// TIA Portal project "PA_test" (V13)

(* hardware
DEVICE "S7300/ET200M station_1"  S7-300 station
   slot 0: "Rail_0"  Rail  6ES7 390-1***0-0AA0
   slot 1: "PS 307 5A_1"  PS 307 5A  6ES7 307-1EA01-0AA0
   slot 2: "PLC-243"  CPU 314C-2 PN/DP  6ES7 314-6EH04-0AB0  V3.3
      slot 2: "PROFINET interface_1"  PN-IO
         slot 1: "Port_1"  Port
         slot 2: "Port_2"  Port
      slot 5: "DI 24/DO 16_1"  DI24/DO16
      slot 6: "AI 5/AO 2_1"  AI5/AO2
      slot 7: "Count_1"  Counter
      slot 8: "Positioning_1"  Positioning
   slot 4: "DI 16x24VDC_1"  DI16 x 24VDC  6ES7 321-1BH02-0AA0
DEVICE "PC station"  SIMATIC PC station
   slot 0: "PC station"  Rail  SIMATIC PC-Station  V1.0
      slot 125: "Stationmanager"  Station_Manager  V6.0.4
   slot 1: "IE general_1"  IE General  IE_CP  V8.2.0
   slot 3: "HMI_RT_1"  WinCC RT Advanced  6AV2 104-0xxxx-xxxx  13.0.1.0
      slot 33792: "Host interface"  Host interface
*)

// ===== PLC "PLC-243"  CPU 314C-2 PN/DP =====

VAR_GLOBAL   // PLC tag table "Default tag table"
   "crna_levo_zgoraj" AT %I1.4 : Bool;
   "crna_desno_zgoraj" AT %I1.6 : Bool;
   "rdeca_levo_zgoraj" AT %Q1.4 : Bool;
   "kljuc" AT %I1.2 : Bool;
   "rdeca_desno_zgoraj" AT %Q1.6 : Bool;
   "stanje" AT %M0.0 : Bool;
   "zelena_tipka" AT %I1.3 : Bool;
   "dvig_smer" AT %Q0.4 : Bool;
   "crna_levo_spodaj" AT %I1.5 : Bool;
   "crna_desno_spodaj" AT %I1.7 : Bool;
   "stevec_trenutno_s" AT %MW4 : Int;
   "miza_premik" AT %Q0.1 : Bool;
   "miza_smer" AT %Q0.0 : Bool;
   "roka_premik" AT %Q0.3 : Bool;
   "roka_smer" AT %Q0.2 : Bool;
   "dvig_premik" AT %Q0.5 : Bool;
   "prijemalo_smer" AT %Q0.6 : Bool;
   "prijemalo_premik" AT %Q0.7 : Bool;
   "koncno_stikalo_miza" AT %I0.0 : Bool;
   "koncno_stikalo_roka" AT %I0.2 : Bool;
   "bit_vrednost" AT %M0.4 : Bool;
   "stevec_impulza_miza" AT %MW10 : Int;
   "impulz_miza" AT %I0.1 : Bool;
   "impulz_roka" AT %I0.3 : Bool;
   "stevec_impulza_roka" AT %MW12 : Int;
   "stevec_impulza_dvig" AT %MW14 : Int;
   "koncno_stikalo_dvig" AT %I0.4 : Bool;
   "impulz_dvig" AT %I0.5 : Bool;
   "koncno_stikalo_prijemalo" AT %I0.6 : Bool;
   "impulz_prijemalo" AT %I0.7 : Bool;
   "stevec_impulza_prijemalo" AT %MW16 : Int;
   "avto_miza_CW" AT %M5.5 : Bool;
   "avto_miza_CCW" AT %M5.6 : Bool;
   "konec_miza" AT %M7.0 : Bool;
   "avto_roka_CW" AT %M5.7 : Bool;
   "avto_roka_CCW" AT %M6.0 : Bool;
   "konec_roka" AT %M6.1 : Bool;
   "avto_dvig_CW" AT %M6.2 : Bool;
   "avto_dvig_CCW" AT %M6.3 : Bool;
   "konec_dvig" AT %M6.4 : Bool;
   "avto_prijemalo_CW" AT %M6.5 : Bool;
   "avto_prijemalo_CCW" AT %M6.6 : Bool;
   "konec_prijemalo" AT %M6.7 : Bool;
   "miza_enable" AT %M7.1 : Bool;
   "miza_koliko" AT %MW8 : Int;
   "roka_koliko" AT %MW18 : Int;
   "dvig_koliko" AT %MW20 : Int;
   "prijemalo_koliko" AT %MW22 : Int;
   "roka_enable" AT %M7.2 : Bool;
   "dvig_enable" AT %M7.3 : Bool;
   "prijemalo_enable" AT %M7.4 : Bool;
   "upravljanje_avtomatov_enable" AT %M24.0 : Bool;
   "rumena_levo_spodaj" AT %Q1.5 : Bool;
   "rumena_desno_spodaj" AT %Q1.7 : Bool;
   "recept" AT %M24.1 : Bool;
END_VAR

TYPE "UDT_lokacija"
   STRUCT
      ID_lokacije : Int;
      miza_lokacija : Int;
      izteg_lokacija : Int;
      stisk_lokacija : Int;
      dvig_lokacija : Int;
   END_STRUCT;
END_TYPE

DATA_BLOCK "stevec_izbira_motorja_DB"   // DB1
{ S7_Optimized_Access := 'FALSE' }
VERSION : 0.1
// stored: InstanceOfName stevec_izbira_motorja
"stevec_izbira_motorja"
BEGIN
END_DATA_BLOCK

DATA_BLOCK "motor_roka"   // DB2
{ S7_Optimized_Access := 'FALSE' }
VERSION : 0.1
// stored: InstanceOfName motor1
"motor1"
BEGIN
END_DATA_BLOCK

DATA_BLOCK "motor1_DB"   // DB3
{ S7_Optimized_Access := 'FALSE' }
VERSION : 0.1
// stored: InstanceOfName motor1
"motor1"
BEGIN
END_DATA_BLOCK

DATA_BLOCK "avtomat_miza_DB"   // DB4
{ S7_Optimized_Access := 'FALSE' }
VERSION : 0.1
// stored: InstanceOfName avtomat_miza
"avtomat_miza"
BEGIN
END_DATA_BLOCK

DATA_BLOCK "Lokacije"   // DB5
{ S7_Optimized_Access := 'FALSE' }
VERSION : 0.1
   VAR
      Lokacija : Array[0..7] of "UDT_lokacija";
   END_VAR
BEGIN
END_DATA_BLOCK

DATA_BLOCK "motor_miza"   // DB6
{ S7_Optimized_Access := 'FALSE' }
VERSION : 0.1
// stored: InstanceOfName motor1
"motor1"
BEGIN
END_DATA_BLOCK

DATA_BLOCK "motor_dvig"   // DB8
{ S7_Optimized_Access := 'FALSE' }
VERSION : 0.1
// stored: InstanceOfName motor1
"motor1"
BEGIN
END_DATA_BLOCK

DATA_BLOCK "motor_prijemalo"   // DB9
{ S7_Optimized_Access := 'FALSE' }
VERSION : 0.1
// stored: InstanceOfName motor1
"motor1"
BEGIN
END_DATA_BLOCK

DATA_BLOCK "avtomat_roka_DB"   // DB10
{ S7_Optimized_Access := 'FALSE' }
VERSION : 0.1
// stored: InstanceOfName avtomat_roka
"avtomat_roka"
BEGIN
END_DATA_BLOCK

DATA_BLOCK "avtomat_dvig_DB"   // DB11
{ S7_Optimized_Access := 'FALSE' }
VERSION : 0.1
// stored: InstanceOfName avtomat_dvig
"avtomat_dvig"
BEGIN
END_DATA_BLOCK

DATA_BLOCK "avtomat_prijemalo_DB"   // DB12
{ S7_Optimized_Access := 'FALSE' }
VERSION : 0.1
// stored: InstanceOfName avtomat_prijemalo
"avtomat_prijemalo"
BEGIN
END_DATA_BLOCK

DATA_BLOCK "upravljanje_avtomatov_DB"   // DB13
{ S7_Optimized_Access := 'FALSE' }
VERSION : 0.1
// stored: InstanceOfName upravljanje_avtomatov
"upravljanje_avtomatov"
BEGIN
END_DATA_BLOCK

DATA_BLOCK "zunanji_krmilnik_DB"   // DB14
{ S7_Optimized_Access := 'FALSE' }
VERSION : 0.1
// stored: InstanceOfName zunanji_krmilnik
"zunanji_krmilnik"
BEGIN
END_DATA_BLOCK

DATA_BLOCK "Lokacije2"   // DB15
{ S7_Optimized_Access := 'FALSE' }
VERSION : 0.1
   VAR
      Lokacija2 : Array[0..7] of "UDT_lokacija";
   END_VAR
BEGIN
END_DATA_BLOCK

DATA_BLOCK "Scada"   // DB16
{ S7_Optimized_Access := 'FALSE' }
VERSION : 0.1
   VAR
      Alarm : Array[1..16] of Bool;
      miza_warning : Bool;
      dvig_warning : Bool;
      prijemalo_warning : Bool;
      roka_warning : Bool;
      Alarm_aktiven : Bool;
      miza_error : Bool;
      dvig_error : Bool;
      prijemalo_error : Bool;
      roka_error : Bool;
      Potrjevanje_alarmov : Bool;
   END_VAR
BEGIN
END_DATA_BLOCK

FUNCTION_BLOCK "motor1"   // FB1, LAD
{ S7_Optimized_Access := 'FALSE' }
VERSION : 0.1
BEGIN

REGION Network 1
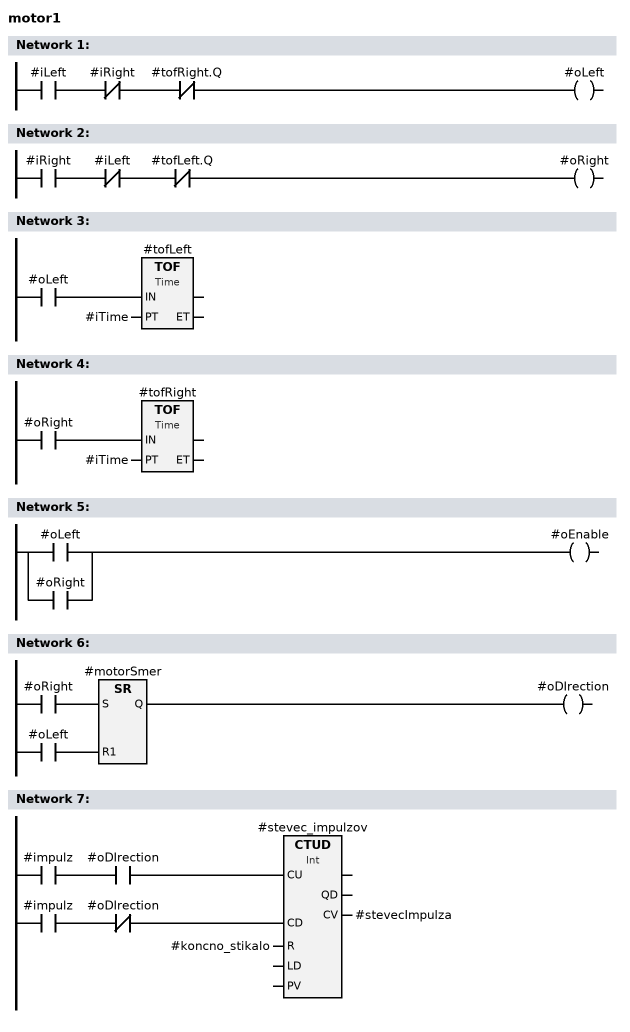
   RUNG wire#powerrail
      Contact( #iLeft )
      I_Contact( #iRight )
      I_Contact( #tofRight.Q )
      Coil( #oLeft )
   END_RUNG
   // the same network as SCL:
   #oLeft := #iLeft AND NOT #iRight AND NOT #tofRight.Q;
END_REGION

REGION Network 2
   RUNG wire#powerrail
      Contact( #iRight )
      I_Contact( #iLeft )
      I_Contact( #tofLeft.Q )
      Coil( #oRight )
   END_RUNG
   // the same network as SCL:
   #oRight := #iRight AND NOT #iLeft AND NOT #tofLeft.Q;
END_REGION

REGION Network 3
   #tofLeft.TOF(IN := #oLeft, PT := #iTime);
END_REGION

REGION Network 4
   #tofRight.TOF(IN := #oRight, PT := #iTime);
END_REGION

REGION Network 5
   RUNG wire#powerrail
      Contact( #oLeft )
      wire#w1
      Coil( #oEnable )
   END_RUNG
   RUNG wire#powerrail
      Contact( #oRight )
   END_RUNG wire#w1
   // the same network as SCL:
   #oEnable := #oLeft OR #oRight;
END_REGION

REGION Network 6
   RUNG wire#powerrail
      Contact( #oRight )
      S_SR(operand := #motorSmer, r1 := wire#w1)
      Coil( #oDIrection )
   END_RUNG
   RUNG wire#powerrail
      Contact( #oLeft )
   END_RUNG wire#w1
   // the same network as SCL:
   IF #oRight THEN
       #motorSmer := TRUE;   // SR flip-flop
   END_IF;
   IF #oLeft THEN #motorSmer := FALSE; END_IF;
   #oDIrection := #motorSmer;
END_REGION

REGION Network 7
   #stevec_impulzov.CTUD(CU := #impulz AND #oDIrection,
                         CD := #impulz AND NOT #oDIrection,
                         R := #koncno_stikalo,
                         CV => #stevecImpulza);
END_REGION
END_FUNCTION_BLOCK

FUNCTION_BLOCK "stevec_izbira_motorja"   // FB2, LAD
{ S7_Optimized_Access := 'FALSE' }
VERSION : 0.1
BEGIN

REGION Network 1
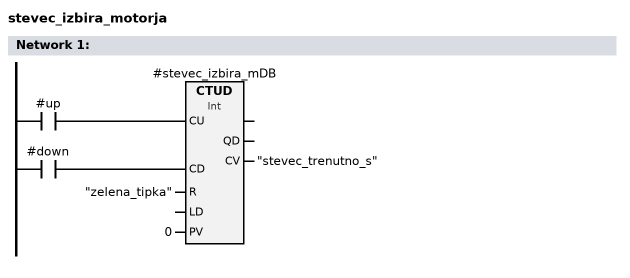
   #stevec_izbira_mDB.CTUD(CU := #up, CD := #down, R := "zelena_tipka", PV := 0, CV => "stevec_trenutno_s");
END_REGION
END_FUNCTION_BLOCK

FUNCTION_BLOCK "avtomat_miza"   // FB3, SCL
{ S7_Optimized_Access := 'FALSE' }
VERSION : 0.1
BEGIN
   IF "Scada".Potrjevanje_alarmov AND "Scada".miza_error THEN
       "Scada".miza_error := 0;
   END_IF;


   IF #enable = TRUE THEN

       IF "motor_miza".stevecImpulza < -40 THEN
           "Scada".miza_warning := 1;
       ELSE
           "Scada".miza_warning := 0;
       END_IF;

       IF #stevilo_premikov < -160 THEN
           "Scada".miza_error := 1;
       ELSE
           "Scada".miza_error := 0;
       END_IF;


       IF #stevilo_premikov <> "motor_miza".stevecImpulza THEN
           IF #stevilo_premikov < "motor_miza".stevecImpulza THEN
               #output_cw := 1;
               #output_ccw := 0;
               #konec_miza := 0;
           END_IF;
           IF #stevilo_premikov > "motor_miza".stevecImpulza THEN
               #output_ccw := 1;
               #output_cw := 0;
               #konec_miza := 0;
           END_IF;
           IF "motor_miza".stevecImpulza - 1 <= #stevilo_premikov AND #stevilo_premikov <= "motor_miza".stevecImpulza + 1 THEN
               #output_cw := 0;
               #output_ccw := 0;
               #konec_miza := 1;
           END_IF;
       END_IF;
       IF #stevilo_premikov = 0 THEN
           IF #stevilo_premikov = "motor_miza".stevecImpulza OR "koncno_stikalo_miza" THEN
               #output_cw := 0;
               #output_ccw := 0;
               #konec_miza := 1;
           ELSE
               #output_ccw := 1;
               #output_cw := 0;
               #konec_miza := 0;
           END_IF;
       END_IF;


   ELSIF #enable = FALSE THEN
       #output_cw := 0;
       #output_ccw := 0;
       #konec_miza := 0;
   END_IF;
END_FUNCTION_BLOCK

FUNCTION_BLOCK "upravljanje_avtomatov"   // FB4, SCL
{ S7_Optimized_Access := 'FALSE' }
VERSION : 0.1
BEGIN
   IF #enable_signal = TRUE THEN
       #miza_enable := 1;
       #roka_enable := 1;
       #dvig_enable := 1;
       #prijemalo_enable := 1;
       #miza_koliko := #lokacija.miza_lokacija;
       #roka_koliko := #lokacija.izteg_lokacija;
       #dvig_koliko := #lokacija.dvig_lokacija;
       #prijemalo_koliko := #lokacija.stisk_lokacija;
   ELSIF #enable_signal = FALSE THEN
       #miza_enable := 0;
       #roka_enable := 0;
       #dvig_enable := 0;
       #prijemalo_enable := 0;
   END_IF;
END_FUNCTION_BLOCK

FUNCTION_BLOCK "avtomat_roka"   // FB5, SCL
{ S7_Optimized_Access := 'FALSE' }
VERSION : 0.1
BEGIN
   IF "Scada".Potrjevanje_alarmov AND "Scada".roka_error THEN
       "Scada".roka_error := 0;
   END_IF;

   IF #enable = TRUE THEN

       IF "motor_roka".stevecImpulza < -40 THEN
           "Scada".roka_warning := 1;
       ELSE
           "Scada".roka_warning := 0;
       END_IF;

       IF #stevilo_premikov < -65 THEN
           "Scada".roka_error := 1;
       ELSE
           "Scada".roka_error := 0;
       END_IF;


       IF #stevilo_premikov <> "motor_roka".stevecImpulza THEN
           IF "motor_roka".stevecImpulza > #stevilo_premikov THEN
               #output_cw := 1;
               #output_ccw := 0;
               #konec_roka := 0;
           END_IF;
           IF "motor_roka".stevecImpulza < #stevilo_premikov THEN
               #output_ccw := 1;
               #output_cw := 0;
               #konec_roka := 0;
           END_IF;
           IF "motor_roka".stevecImpulza - 1 <= #stevilo_premikov AND #stevilo_premikov <= "motor_roka".stevecImpulza + 1 THEN
               #output_cw := 0;
               #output_ccw := 0;
               #konec_roka := 1;
           END_IF;
       END_IF;
       IF #stevilo_premikov = 0 THEN
           IF #stevilo_premikov = "motor_roka".stevecImpulza OR "koncno_stikalo_roka" THEN
               #output_cw := 0;
               #output_ccw := 0;
               #konec_roka := 1;
           ELSE
               #output_ccw := 1;
               #output_cw := 0;
               #konec_roka := 0;
           END_IF;
       END_IF;

   ELSIF #enable = FALSE THEN
       #output_cw := 0;
       #output_ccw := 0;
       #konec_roka := 0;
   END_IF;
END_FUNCTION_BLOCK

FUNCTION_BLOCK "avtomat_dvig"   // FB6, SCL
{ S7_Optimized_Access := 'FALSE' }
VERSION : 0.1
BEGIN
   IF "Scada".Potrjevanje_alarmov AND "Scada".dvig_error THEN
       "Scada".dvig_error := 0;
   END_IF;



   IF #enable = TRUE THEN

       IF "motor_dvig".stevecImpulza > 100 THEN
           "Scada".dvig_warning := 1;
       ELSE
           "Scada".dvig_warning := 0;
       END_IF;

       IF #stevilo_premikov > 115 THEN
           "Scada".dvig_error := 1;
       ELSE
           "Scada".dvig_error := 0;
       END_IF;

       IF #stevilo_premikov <> "motor_dvig".stevecImpulza THEN
           IF "motor_dvig".stevecImpulza > #stevilo_premikov THEN
               #output_cw := 1;
               #output_ccw := 0;
               #konec_dvig := 0;
           END_IF;
           IF "motor_dvig".stevecImpulza < #stevilo_premikov THEN
               #output_ccw := 1;
               #output_cw := 0;
               #konec_dvig := 0;
           END_IF;
           IF "motor_dvig".stevecImpulza - 1 <= #stevilo_premikov AND #stevilo_premikov <= "motor_dvig".stevecImpulza + 1 THEN
               #output_cw := 0;
               #output_ccw := 0;
               #konec_dvig := 1;
           END_IF;
       END_IF;
       IF #stevilo_premikov = 0 THEN
           IF #stevilo_premikov = "motor_dvig".stevecImpulza OR "koncno_stikalo_dvig" THEN
               #output_cw := 0;
               #output_ccw := 0;
               #konec_dvig := 1;
           ELSE
               #output_cw := 1;
               #output_ccw := 0;
               #konec_dvig := 0;
           END_IF;
       END_IF;
   ELSIF #enable = FALSE THEN
       #output_cw := 0;
       #output_ccw := 0;
       #konec_dvig := 0;
   END_IF;
END_FUNCTION_BLOCK

FUNCTION_BLOCK "avtomat_prijemalo"   // FB7, SCL
{ S7_Optimized_Access := 'FALSE' }
VERSION : 0.1
BEGIN
   IF "Scada".Potrjevanje_alarmov AND "Scada".prijemalo_error THEN
       "Scada".prijemalo_error := 0;
   END_IF;



   IF #enable = TRUE THEN

       IF "motor_prijemalo".stevecImpulza > 10 THEN
           "Scada".prijemalo_warning := 1;
       ELSE
           "Scada".prijemalo_warning := 0;
       END_IF;

       IF #stevilo_premikov > 15 THEN
           "Scada".prijemalo_error := 1;
       ELSE
           "Scada".prijemalo_error := 0;
       END_IF;

       IF #stevilo_premikov <> "motor_prijemalo".stevecImpulza THEN
           IF "motor_prijemalo".stevecImpulza > #stevilo_premikov THEN
               #output_cw := 1;
               #output_ccw := 0;
               #konec_prijemalo := 0;
           END_IF;
           IF "motor_prijemalo".stevecImpulza < #stevilo_premikov THEN
               #output_ccw := 1;
               #output_cw := 0;
               #konec_prijemalo := 0;
           END_IF;
           IF "motor_prijemalo".stevecImpulza - 1 <= #stevilo_premikov AND #stevilo_premikov <= "motor_prijemalo".stevecImpulza + 1 THEN
               #output_cw := 0;
               #output_ccw := 0;
               #konec_prijemalo := 1;
           END_IF;
       END_IF;
       IF #stevilo_premikov = 0 THEN
           IF #stevilo_premikov = "motor_prijemalo".stevecImpulza OR "koncno_stikalo_prijemalo" THEN
               #output_cw := 0;
               #output_ccw := 0;
               #konec_prijemalo := 1;
           ELSE
               #output_cw := 1;
               #output_ccw := 0;
               #konec_prijemalo := 0;
           END_IF;
       END_IF;


   ELSIF #enable = FALSE THEN
       #output_cw := 0;
       #output_ccw := 0;
       #konec_prijemalo := 0;
   END_IF;
END_FUNCTION_BLOCK

FUNCTION_BLOCK "zunanji_krmilnik"   // FB8, SCL
{ S7_Optimized_Access := 'FALSE' }
VERSION : 0.1
BEGIN

   IF "Scada".Potrjevanje_alarmov AND "Scada".miza_error = 0 AND "Scada".dvig_error = 0 AND "Scada".roka_error = 0 AND "Scada".prijemalo_error = 0 THEN
       #upravljanje_avtomatov_enable := TRUE;
       "Scada".Potrjevanje_alarmov := FALSE;
   END_IF;

   IF #enable  THEN
       IF "recept" = 0 THEN
           IF #trenutni_index < #stevilo_lokacij AND "Scada".miza_error = 0 AND "Scada".dvig_error = 0 AND "Scada".roka_error = 0 AND "Scada".prijemalo_error = 0 THEN
               #upravljanje_avtomatov_enable := TRUE;
               #naslednja_lokacija := #Lokacija[#trenutni_index];
           ELSE
               #upravljanje_avtomatov_enable := FALSE;
           END_IF;
       END_IF;
       IF "avtomat_miza_DB".konec_miza AND "avtomat_dvig_DB".konec_dvig AND "avtomat_roka_DB".konec_roka AND "avtomat_prijemalo_DB".konec_prijemalo AND #povecaj_index = 1 THEN
           #trenutni_index := #trenutni_index + 1;
           #povecaj_index := 0;
       ELSE
           #povecaj_index := 1;
       END_IF;
       IF #trenutni_index = #stevilo_lokacij THEN
           #trenutni_index := 0;
       END_IF;

       IF "recept" = 1 THEN
           IF #trenutni_index2 < #stevilo_lokacij AND "Scada".miza_error = 0 AND "Scada".dvig_error = 0 AND "Scada".roka_error = 0 AND "Scada".prijemalo_error = 0 THEN
               #upravljanje_avtomatov_enable := TRUE;
               #naslednja_lokacija := #Lokacija2[#trenutni_index2];
           ELSE
               #upravljanje_avtomatov_enable := FALSE;
           END_IF;
       END_IF;
       IF "avtomat_miza_DB".konec_miza AND "avtomat_dvig_DB".konec_dvig AND "avtomat_roka_DB".konec_roka AND "avtomat_prijemalo_DB".konec_prijemalo AND #povecaj_index2 = 1 THEN
           #trenutni_index2 := #trenutni_index2 + 1;
           #povecaj_index2 := 0;
       ELSE
           #povecaj_index2 := 1;
       END_IF;
       IF #trenutni_index2 = #stevilo_lokacij THEN
           #trenutni_index2 := 0;
       END_IF;

   ELSIF #enable = FALSE THEN
       #upravljanje_avtomatov_enable := FALSE;
       #povecaj_index := 0;
       #povecaj_index2 := 0;
   END_IF;
END_FUNCTION_BLOCK

FUNCTION "reset_funkcija" : Void   // FC1, SCL
{ S7_Optimized_Access := 'FALSE' }
VERSION : 0.1
BEGIN
   IF #zelena_tipka THEN
       "Scada".miza_error := 0;
       "Scada".roka_error := 0;
       "Scada".dvig_error := 0;
       "Scada".prijemalo_error := 0;

       "zunanji_krmilnik_DB".naslednja_lokacija.ID_lokacije := 0;
       "zunanji_krmilnik_DB".naslednja_lokacija.miza_lokacija := 0;
       "zunanji_krmilnik_DB".naslednja_lokacija.izteg_lokacija := 0;
       "zunanji_krmilnik_DB".naslednja_lokacija.stisk_lokacija := 0;
       "zunanji_krmilnik_DB".naslednja_lokacija.dvig_lokacija := 0;

       "zunanji_krmilnik_DB".trenutni_index := 0;
       "zunanji_krmilnik_DB".trenutni_index2 := 0;


   END_IF;
END_FUNCTION

FUNCTION "Alarmi" : Void   // FC2, LAD
{ S7_Optimized_Access := 'FALSE' }
VERSION : 0.1
BEGIN

REGION Network 1: miza opozorilo
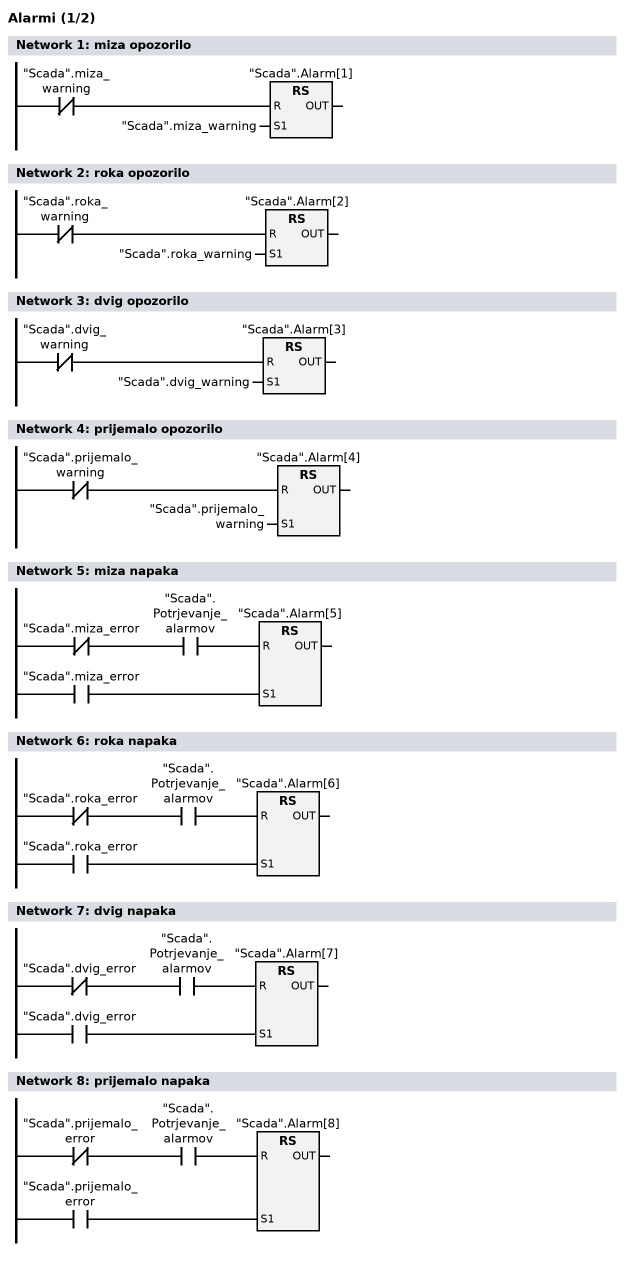
   RUNG wire#powerrail
      I_Contact( "Scada".miza_warning )
      S_RS(operand := "Scada".Alarm[1], s1 := "Scada".miza_warning)
   END_RUNG
   // the same network as SCL:
   IF NOT "Scada".miza_warning THEN
       "Scada".Alarm[1] := FALSE;   // RS flip-flop
   END_IF;
   IF "Scada".miza_warning THEN "Scada".Alarm[1] := TRUE; END_IF;
END_REGION

REGION Network 2: roka opozorilo
   RUNG wire#powerrail
      I_Contact( "Scada".roka_warning )
      S_RS(operand := "Scada".Alarm[2], s1 := "Scada".roka_warning)
   END_RUNG
   // the same network as SCL:
   IF NOT "Scada".roka_warning THEN
       "Scada".Alarm[2] := FALSE;   // RS flip-flop
   END_IF;
   IF "Scada".roka_warning THEN "Scada".Alarm[2] := TRUE; END_IF;
END_REGION

REGION Network 3: dvig opozorilo
   RUNG wire#powerrail
      I_Contact( "Scada".dvig_warning )
      S_RS(operand := "Scada".Alarm[3], s1 := "Scada".dvig_warning)
   END_RUNG
   // the same network as SCL:
   IF NOT "Scada".dvig_warning THEN
       "Scada".Alarm[3] := FALSE;   // RS flip-flop
   END_IF;
   IF "Scada".dvig_warning THEN "Scada".Alarm[3] := TRUE; END_IF;
END_REGION

REGION Network 4: prijemalo opozorilo
   RUNG wire#powerrail
      I_Contact( "Scada".prijemalo_warning )
      S_RS(operand := "Scada".Alarm[4], s1 := "Scada".prijemalo_warning)
   END_RUNG
   // the same network as SCL:
   IF NOT "Scada".prijemalo_warning THEN
       "Scada".Alarm[4] := FALSE;   // RS flip-flop
   END_IF;
   IF "Scada".prijemalo_warning THEN "Scada".Alarm[4] := TRUE; END_IF;
END_REGION

REGION Network 5: miza napaka
   RUNG wire#powerrail
      I_Contact( "Scada".miza_error )
      Contact( "Scada".Potrjevanje_alarmov )
      S_RS(operand := "Scada".Alarm[5], s1 := wire#w1)
   END_RUNG
   RUNG wire#powerrail
      Contact( "Scada".miza_error )
   END_RUNG wire#w1
   // the same network as SCL:
   IF NOT "Scada".miza_error AND "Scada".Potrjevanje_alarmov THEN
       "Scada".Alarm[5] := FALSE;   // RS flip-flop
   END_IF;
   IF "Scada".miza_error THEN "Scada".Alarm[5] := TRUE; END_IF;
END_REGION

REGION Network 6: roka napaka
   RUNG wire#powerrail
      I_Contact( "Scada".roka_error )
      Contact( "Scada".Potrjevanje_alarmov )
      S_RS(operand := "Scada".Alarm[6], s1 := wire#w1)
   END_RUNG
   RUNG wire#powerrail
      Contact( "Scada".roka_error )
   END_RUNG wire#w1
   // the same network as SCL:
   IF NOT "Scada".roka_error AND "Scada".Potrjevanje_alarmov THEN
       "Scada".Alarm[6] := FALSE;   // RS flip-flop
   END_IF;
   IF "Scada".roka_error THEN "Scada".Alarm[6] := TRUE; END_IF;
END_REGION

REGION Network 7: dvig napaka
   RUNG wire#powerrail
      I_Contact( "Scada".dvig_error )
      Contact( "Scada".Potrjevanje_alarmov )
      S_RS(operand := "Scada".Alarm[7], s1 := wire#w1)
   END_RUNG
   RUNG wire#powerrail
      Contact( "Scada".dvig_error )
   END_RUNG wire#w1
   // the same network as SCL:
   IF NOT "Scada".dvig_error AND "Scada".Potrjevanje_alarmov THEN
       "Scada".Alarm[7] := FALSE;   // RS flip-flop
   END_IF;
   IF "Scada".dvig_error THEN "Scada".Alarm[7] := TRUE; END_IF;
END_REGION

REGION Network 8: prijemalo napaka
   RUNG wire#powerrail
      I_Contact( "Scada".prijemalo_error )
      Contact( "Scada".Potrjevanje_alarmov )
      S_RS(operand := "Scada".Alarm[8], s1 := wire#w1)
   END_RUNG
   RUNG wire#powerrail
      Contact( "Scada".prijemalo_error )
   END_RUNG wire#w1
   // the same network as SCL:
   IF NOT "Scada".prijemalo_error AND "Scada".Potrjevanje_alarmov THEN
       "Scada".Alarm[8] := FALSE;   // RS flip-flop
   END_IF;
   IF "Scada".prijemalo_error THEN "Scada".Alarm[8] := TRUE; END_IF;
END_REGION

REGION Network 9: info premikanje avto
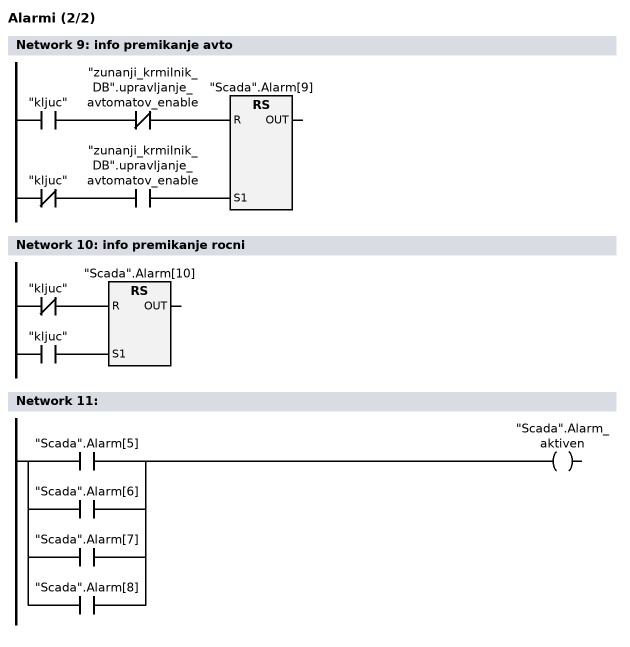
   RUNG wire#powerrail
      Contact( "kljuc" )
      I_Contact( "zunanji_krmilnik_DB".upravljanje_avtomatov_enable )
      S_RS(operand := "Scada".Alarm[9], s1 := wire#w1)
   END_RUNG
   RUNG wire#powerrail
      I_Contact( "kljuc" )
      Contact( "zunanji_krmilnik_DB".upravljanje_avtomatov_enable )
   END_RUNG wire#w1
   // the same network as SCL:
   IF "kljuc" AND NOT "zunanji_krmilnik_DB".upravljanje_avtomatov_enable THEN
       "Scada".Alarm[9] := FALSE;   // RS flip-flop
   END_IF;
   IF NOT "kljuc" AND "zunanji_krmilnik_DB".upravljanje_avtomatov_enable THEN
       "Scada".Alarm[9] := TRUE;
   END_IF;
END_REGION

REGION Network 10: info premikanje rocni
   RUNG wire#powerrail
      I_Contact( "kljuc" )
      S_RS(operand := "Scada".Alarm[10], s1 := wire#w1)
   END_RUNG
   RUNG wire#powerrail
      Contact( "kljuc" )
   END_RUNG wire#w1
   // the same network as SCL:
   IF NOT "kljuc" THEN
       "Scada".Alarm[10] := FALSE;   // RS flip-flop
   END_IF;
   IF "kljuc" THEN "Scada".Alarm[10] := TRUE; END_IF;
END_REGION

REGION Network 11
   RUNG wire#powerrail
      Contact( "Scada".Alarm[5] )
      wire#w1
      Coil( "Scada".Alarm_aktiven )
   END_RUNG
   RUNG wire#powerrail
      Contact( "Scada".Alarm[6] )
   END_RUNG wire#w1
   RUNG wire#powerrail
      Contact( "Scada".Alarm[7] )
   END_RUNG wire#w1
   RUNG wire#powerrail
      Contact( "Scada".Alarm[8] )
   END_RUNG wire#w1
   // the same network as SCL:
   "Scada".Alarm_aktiven := "Scada".Alarm[5] OR "Scada".Alarm[6] OR "Scada".Alarm[7] OR "Scada".Alarm[8];
END_REGION
END_FUNCTION

ORGANIZATION_BLOCK "Main"   // OB1, LAD
TITLE = "Main Program Sweep (Cycle)"
{ S7_Optimized_Access := 'FALSE' }
VERSION : 0.1
BEGIN

REGION Network 1: alarmi
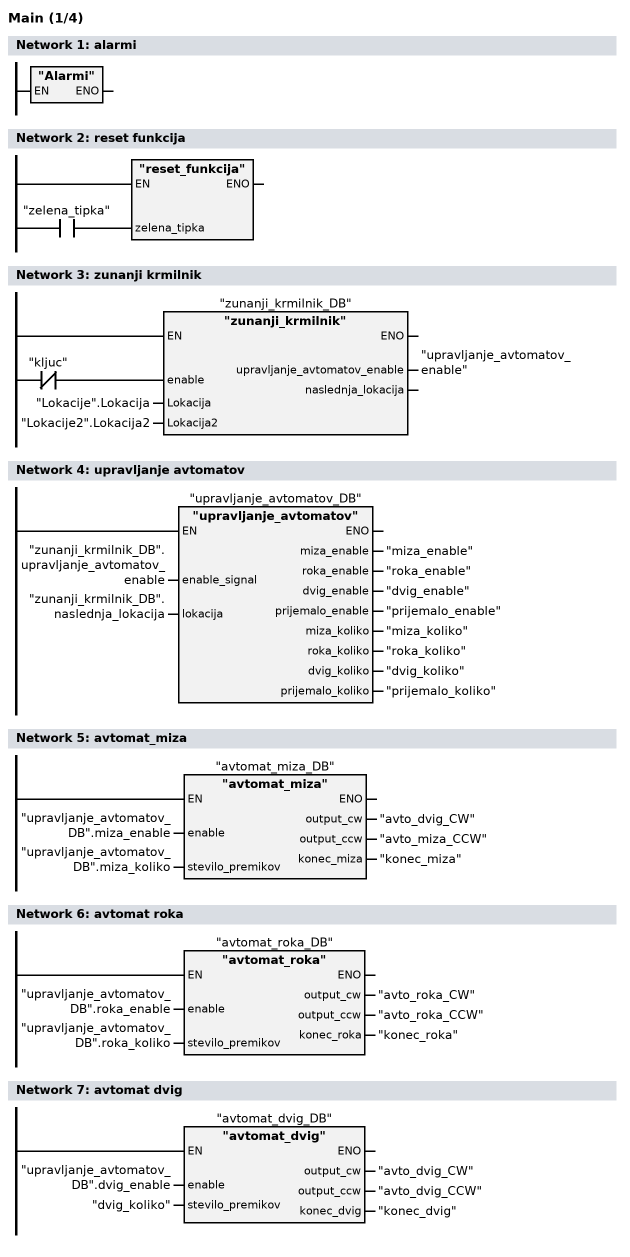
   RUNG wire#powerrail
      "Alarmi"()
   END_RUNG
   // the same network as SCL:
   "Alarmi"();
END_REGION

REGION Network 2: reset funkcija
   RUNG wire#powerrail
      "reset_funkcija"(zelena_tipka := wire#w1)
   END_RUNG
   RUNG wire#powerrail
      Contact( "zelena_tipka" )
   END_RUNG wire#w1
   // the same network as SCL:
   "reset_funkcija"(zelena_tipka := "zelena_tipka");
END_REGION

REGION Network 3: zunanji krmilnik
   RUNG wire#powerrail
      "zunanji_krmilnik_DB"(enable := wire#w1, Lokacija := "Lokacije".Lokacija, Lokacija2 := "Lokacije2".Lokacija2, upravljanje_avtomatov_enable => "upravljanje_avtomatov_enable", naslednja_lokacija =>)
   END_RUNG
   RUNG wire#powerrail
      I_Contact( "kljuc" )
   END_RUNG wire#w1
   // the same network as SCL:
   "zunanji_krmilnik_DB"(enable := NOT "kljuc",   // "zunanji_krmilnik"
                         Lokacija := "Lokacije".Lokacija,
                         Lokacija2 := "Lokacije2".Lokacija2,
                         upravljanje_avtomatov_enable => "upravljanje_avtomatov_enable");
END_REGION

REGION Network 4: upravljanje avtomatov
   RUNG wire#powerrail
      "upravljanje_avtomatov_DB"(enable_signal := "zunanji_krmilnik_DB".upravljanje_avtomatov_enable, lokacija := "zunanji_krmilnik_DB".naslednja_lokacija, miza_enable => "miza_enable", roka_enable => "roka_enable", dvig_enable => "dvig_enable", prijemalo_enable => "prijemalo_enable", miza_koliko => "miza_koliko", roka_koliko => "roka_koliko", dvig_koliko => "dvig_koliko", prijemalo_koliko => "prijemalo_koliko")
   END_RUNG
   // the same network as SCL:
   "upravljanje_avtomatov_DB"(enable_signal := "zunanji_krmilnik_DB".upravljanje_avtomatov_enable,   // "upravljanje_avtomatov"
                           lokacija := "zunanji_krmilnik_DB".naslednja_lokacija,
                           miza_enable => "miza_enable",
                           roka_enable => "roka_enable",
                           dvig_enable => "dvig_enable",
                           prijemalo_enable => "prijemalo_enable",
                           miza_koliko => "miza_koliko",
                           roka_koliko => "roka_koliko",
                           dvig_koliko => "dvig_koliko",
                           prijemalo_koliko => "prijemalo_koliko");
END_REGION

REGION Network 5: avtomat_miza
   RUNG wire#powerrail
      "avtomat_miza_DB"(enable := "upravljanje_avtomatov_DB".miza_enable, stevilo_premikov := "upravljanje_avtomatov_DB".miza_koliko, output_cw => "avto_dvig_CW", output_ccw => "avto_miza_CCW", konec_miza => "konec_miza")
   END_RUNG
   // the same network as SCL:
   "avtomat_miza_DB"(enable := "upravljanje_avtomatov_DB".miza_enable,   // "avtomat_miza"
                     stevilo_premikov := "upravljanje_avtomatov_DB".miza_koliko,
                     output_cw => "avto_dvig_CW",
                     output_ccw => "avto_miza_CCW",
                     konec_miza => "konec_miza");
END_REGION

REGION Network 6: avtomat roka
   RUNG wire#powerrail
      "avtomat_roka_DB"(enable := "upravljanje_avtomatov_DB".roka_enable, stevilo_premikov := "upravljanje_avtomatov_DB".roka_koliko, output_cw => "avto_roka_CW", output_ccw => "avto_roka_CCW", konec_roka => "konec_roka")
   END_RUNG
   // the same network as SCL:
   "avtomat_roka_DB"(enable := "upravljanje_avtomatov_DB".roka_enable,   // "avtomat_roka"
                     stevilo_premikov := "upravljanje_avtomatov_DB".roka_koliko,
                     output_cw => "avto_roka_CW",
                     output_ccw => "avto_roka_CCW",
                     konec_roka => "konec_roka");
END_REGION

REGION Network 7: avtomat dvig
   RUNG wire#powerrail
      "avtomat_dvig_DB"(enable := "upravljanje_avtomatov_DB".dvig_enable, stevilo_premikov := "dvig_koliko", output_cw => "avto_dvig_CW", output_ccw => "avto_dvig_CCW", konec_dvig => "konec_dvig")
   END_RUNG
   // the same network as SCL:
   "avtomat_dvig_DB"(enable := "upravljanje_avtomatov_DB".dvig_enable,   // "avtomat_dvig"
                     stevilo_premikov := "dvig_koliko",
                     output_cw => "avto_dvig_CW",
                     output_ccw => "avto_dvig_CCW",
                     konec_dvig => "konec_dvig");
END_REGION

REGION Network 8: avtomat prijemalo
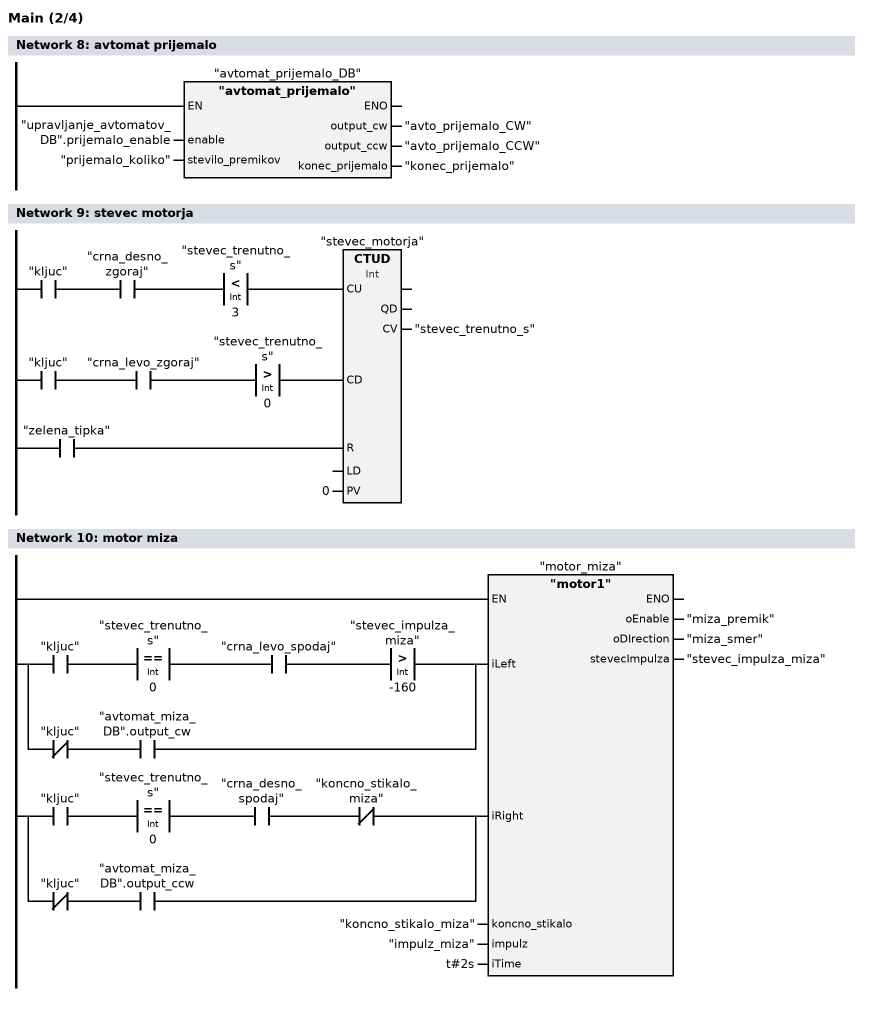
   RUNG wire#powerrail
      "avtomat_prijemalo_DB"(enable := "upravljanje_avtomatov_DB".prijemalo_enable, stevilo_premikov := "prijemalo_koliko", output_cw => "avto_prijemalo_CW", output_ccw => "avto_prijemalo_CCW", konec_prijemalo => "konec_prijemalo")
   END_RUNG
   // the same network as SCL:
   "avtomat_prijemalo_DB"(enable := "upravljanje_avtomatov_DB".prijemalo_enable,   // "avtomat_prijemalo"
                          stevilo_premikov := "prijemalo_koliko",
                          output_cw => "avto_prijemalo_CW",
                          output_ccw => "avto_prijemalo_CCW",
                          konec_prijemalo => "konec_prijemalo");
END_REGION

REGION Network 9: stevec motorja
   "stevec_motorja".CTUD(CU := "kljuc" AND "crna_desno_zgoraj" AND ("stevec_trenutno_s" < 3),
                         CD := "kljuc" AND "crna_levo_zgoraj" AND ("stevec_trenutno_s" > 0),
                         R := "zelena_tipka",
                         PV := 0,
                         CV => "stevec_trenutno_s");
END_REGION

REGION Network 10: motor miza
   RUNG wire#powerrail
      "motor_miza"(iLeft := wire#w1, iRight := wire#w2, koncno_stikalo := "koncno_stikalo_miza", impulz := "impulz_miza", iTime := t#2s, oEnable => "miza_premik", oDIrection => "miza_smer", stevecImpulza => "stevec_impulza_miza")
   END_RUNG
   RUNG wire#powerrail
      Contact( "kljuc" )
      { S7_Templates := "SrcType := Int" } EQ_Contact(in1 := "stevec_trenutno_s", in2 := 0)
      Contact( "crna_levo_spodaj" )
      { S7_Templates := "SrcType := Int" } GT_Contact(in1 := "stevec_impulza_miza", in2 := -160)
   END_RUNG wire#w1
   RUNG wire#powerrail
      I_Contact( "kljuc" )
      Contact( "avtomat_miza_DB".output_cw )
   END_RUNG wire#w1
   RUNG wire#powerrail
      Contact( "kljuc" )
      { S7_Templates := "SrcType := Int" } EQ_Contact(in1 := "stevec_trenutno_s", in2 := 0)
      Contact( "crna_desno_spodaj" )
      I_Contact( "koncno_stikalo_miza" )
   END_RUNG wire#w2
   RUNG wire#powerrail
      I_Contact( "kljuc" )
      Contact( "avtomat_miza_DB".output_ccw )
   END_RUNG wire#w2
   // the same network as SCL:
   "motor_miza"(iLeft := ("kljuc" AND ("stevec_trenutno_s" = 0) AND "crna_levo_spodaj" AND ("stevec_impulza_miza" > (-160))) OR (NOT "kljuc" AND "avtomat_miza_DB".output_cw),   // "motor1"
                iRight := ("kljuc" AND ("stevec_trenutno_s" = 0) AND "crna_desno_spodaj" AND NOT "koncno_stikalo_miza") OR (NOT "kljuc" AND "avtomat_miza_DB".output_ccw),
                koncno_stikalo := "koncno_stikalo_miza",
                impulz := "impulz_miza",
                iTime := t#2s,
                oEnable => "miza_premik",
                oDIrection => "miza_smer",
                stevecImpulza => "stevec_impulza_miza");
END_REGION

REGION Network 11: motor roka
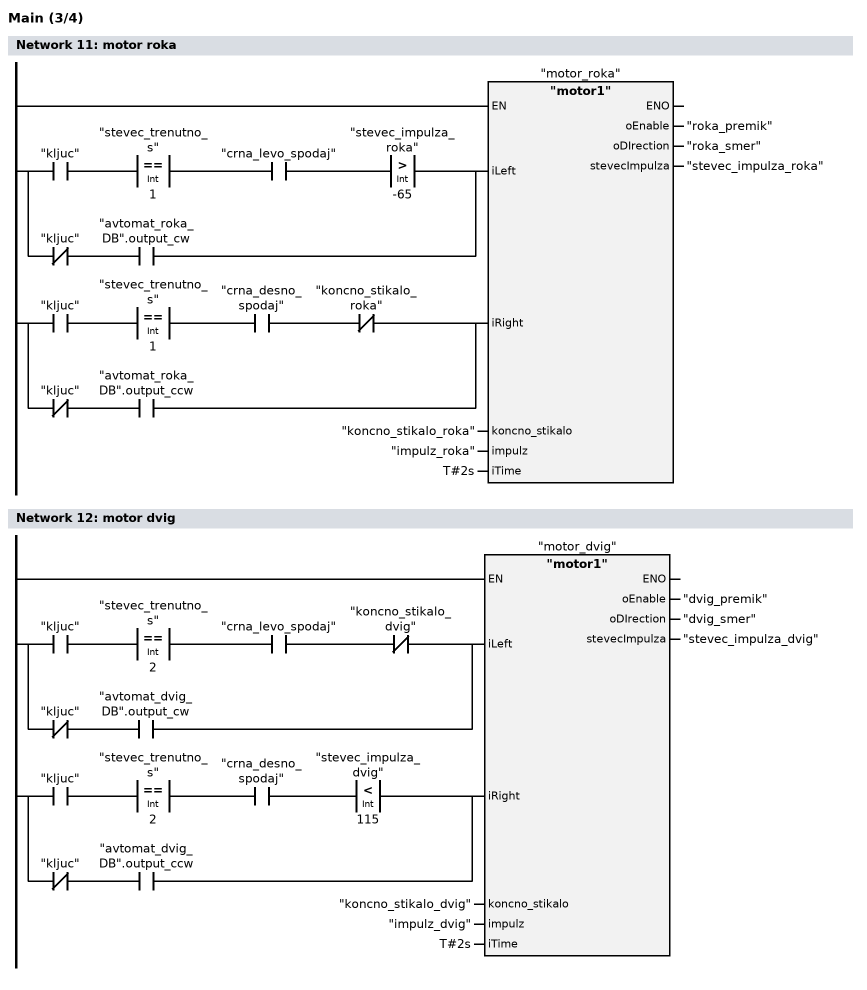
   RUNG wire#powerrail
      "motor_roka"(iLeft := wire#w1, iRight := wire#w2, koncno_stikalo := "koncno_stikalo_roka", impulz := "impulz_roka", iTime := T#2s, oEnable => "roka_premik", oDIrection => "roka_smer", stevecImpulza => "stevec_impulza_roka")
   END_RUNG
   RUNG wire#powerrail
      Contact( "kljuc" )
      { S7_Templates := "SrcType := Int" } EQ_Contact(in1 := "stevec_trenutno_s", in2 := 1)
      Contact( "crna_levo_spodaj" )
      { S7_Templates := "SrcType := Int" } GT_Contact(in1 := "stevec_impulza_roka", in2 := -65)
   END_RUNG wire#w1
   RUNG wire#powerrail
      I_Contact( "kljuc" )
      Contact( "avtomat_roka_DB".output_cw )
   END_RUNG wire#w1
   RUNG wire#powerrail
      Contact( "kljuc" )
      { S7_Templates := "SrcType := Int" } EQ_Contact(in1 := "stevec_trenutno_s", in2 := 1)
      Contact( "crna_desno_spodaj" )
      I_Contact( "koncno_stikalo_roka" )
   END_RUNG wire#w2
   RUNG wire#powerrail
      I_Contact( "kljuc" )
      Contact( "avtomat_roka_DB".output_ccw )
   END_RUNG wire#w2
   // the same network as SCL:
   "motor_roka"(iLeft := ("kljuc" AND ("stevec_trenutno_s" = 1) AND "crna_levo_spodaj" AND ("stevec_impulza_roka" > (-65))) OR (NOT "kljuc" AND "avtomat_roka_DB".output_cw),   // "motor1"
                iRight := ("kljuc" AND ("stevec_trenutno_s" = 1) AND "crna_desno_spodaj" AND NOT "koncno_stikalo_roka") OR (NOT "kljuc" AND "avtomat_roka_DB".output_ccw),
                koncno_stikalo := "koncno_stikalo_roka",
                impulz := "impulz_roka",
                iTime := T#2s,
                oEnable => "roka_premik",
                oDIrection => "roka_smer",
                stevecImpulza => "stevec_impulza_roka");
END_REGION

REGION Network 12: motor dvig
   RUNG wire#powerrail
      "motor_dvig"(iLeft := wire#w1, iRight := wire#w2, koncno_stikalo := "koncno_stikalo_dvig", impulz := "impulz_dvig", iTime := T#2s, oEnable => "dvig_premik", oDIrection => "dvig_smer", stevecImpulza => "stevec_impulza_dvig")
   END_RUNG
   RUNG wire#powerrail
      Contact( "kljuc" )
      { S7_Templates := "SrcType := Int" } EQ_Contact(in1 := "stevec_trenutno_s", in2 := 2)
      Contact( "crna_levo_spodaj" )
      I_Contact( "koncno_stikalo_dvig" )
   END_RUNG wire#w1
   RUNG wire#powerrail
      I_Contact( "kljuc" )
      Contact( "avtomat_dvig_DB".output_cw )
   END_RUNG wire#w1
   RUNG wire#powerrail
      Contact( "kljuc" )
      { S7_Templates := "SrcType := Int" } EQ_Contact(in1 := "stevec_trenutno_s", in2 := 2)
      Contact( "crna_desno_spodaj" )
      { S7_Templates := "SrcType := Int" } LT_Contact(in1 := "stevec_impulza_dvig", in2 := 115)
   END_RUNG wire#w2
   RUNG wire#powerrail
      I_Contact( "kljuc" )
      Contact( "avtomat_dvig_DB".output_ccw )
   END_RUNG wire#w2
   // the same network as SCL:
   "motor_dvig"(iLeft := ("kljuc" AND ("stevec_trenutno_s" = 2) AND "crna_levo_spodaj" AND NOT "koncno_stikalo_dvig") OR (NOT "kljuc" AND "avtomat_dvig_DB".output_cw),   // "motor1"
                iRight := ("kljuc" AND ("stevec_trenutno_s" = 2) AND "crna_desno_spodaj" AND ("stevec_impulza_dvig" < 115)) OR (NOT "kljuc" AND "avtomat_dvig_DB".output_ccw),
                koncno_stikalo := "koncno_stikalo_dvig",
                impulz := "impulz_dvig",
                iTime := T#2s,
                oEnable => "dvig_premik",
                oDIrection => "dvig_smer",
                stevecImpulza => "stevec_impulza_dvig");
END_REGION

REGION Network 13: motor prijemalo
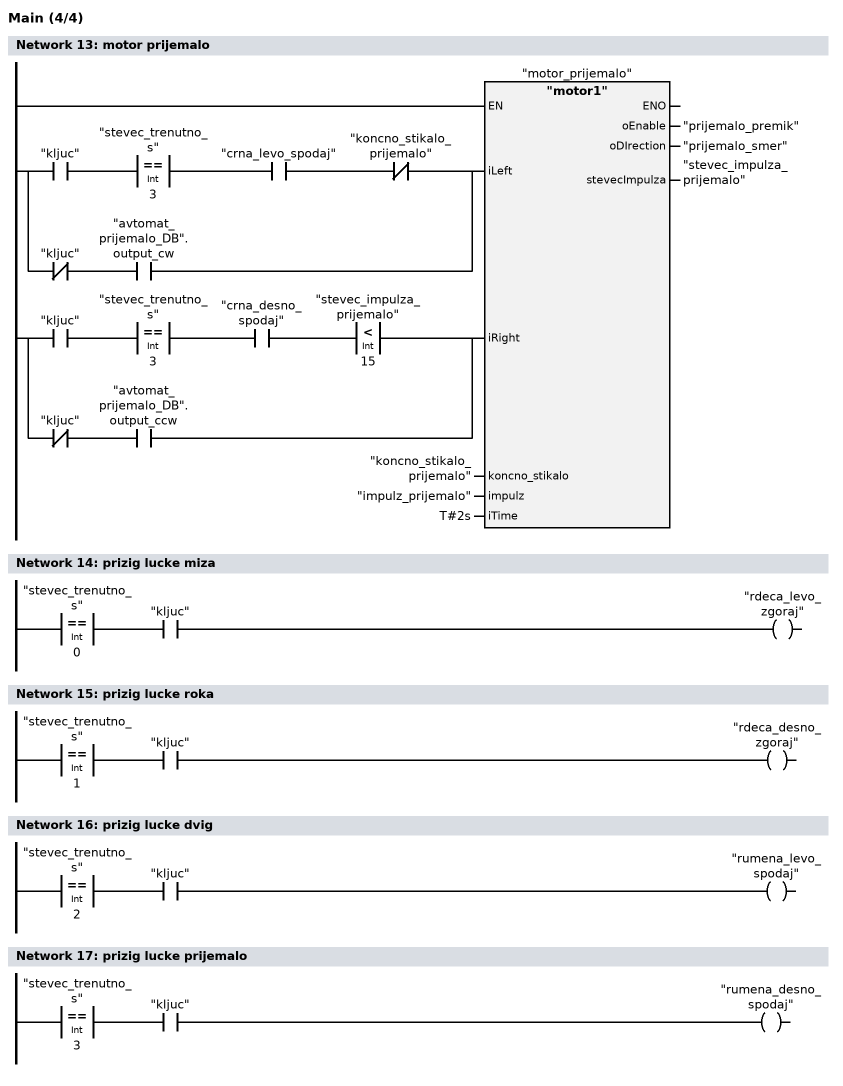
   RUNG wire#powerrail
      "motor_prijemalo"(iLeft := wire#w1, iRight := wire#w2, koncno_stikalo := "koncno_stikalo_prijemalo", impulz := "impulz_prijemalo", iTime := T#2s, oEnable => "prijemalo_premik", oDIrection => "prijemalo_smer", stevecImpulza => "stevec_impulza_prijemalo")
   END_RUNG
   RUNG wire#powerrail
      Contact( "kljuc" )
      { S7_Templates := "SrcType := Int" } EQ_Contact(in1 := "stevec_trenutno_s", in2 := 3)
      Contact( "crna_levo_spodaj" )
      I_Contact( "koncno_stikalo_prijemalo" )
   END_RUNG wire#w1
   RUNG wire#powerrail
      I_Contact( "kljuc" )
      Contact( "avtomat_prijemalo_DB".output_cw )
   END_RUNG wire#w1
   RUNG wire#powerrail
      Contact( "kljuc" )
      { S7_Templates := "SrcType := Int" } EQ_Contact(in1 := "stevec_trenutno_s", in2 := 3)
      Contact( "crna_desno_spodaj" )
      { S7_Templates := "SrcType := Int" } LT_Contact(in1 := "stevec_impulza_prijemalo", in2 := 15)
   END_RUNG wire#w2
   RUNG wire#powerrail
      I_Contact( "kljuc" )
      Contact( "avtomat_prijemalo_DB".output_ccw )
   END_RUNG wire#w2
   // the same network as SCL:
   "motor_prijemalo"(iLeft := ("kljuc" AND ("stevec_trenutno_s" = 3) AND "crna_levo_spodaj" AND NOT "koncno_stikalo_prijemalo") OR (NOT "kljuc" AND "avtomat_prijemalo_DB".output_cw),   // "motor1"
                     iRight := ("kljuc" AND ("stevec_trenutno_s" = 3) AND "crna_desno_spodaj" AND ("stevec_impulza_prijemalo" < 15)) OR (NOT "kljuc" AND "avtomat_prijemalo_DB".output_ccw),
                     koncno_stikalo := "koncno_stikalo_prijemalo",
                     impulz := "impulz_prijemalo",
                     iTime := T#2s,
                     oEnable => "prijemalo_premik",
                     oDIrection => "prijemalo_smer",
                     stevecImpulza => "stevec_impulza_prijemalo");
END_REGION

REGION Network 14: prizig lucke miza
   RUNG wire#powerrail
      { S7_Templates := "SrcType := Int" } EQ_Contact(in1 := "stevec_trenutno_s", in2 := 0)
      Contact( "kljuc" )
      Coil( "rdeca_levo_zgoraj" )
   END_RUNG
   // the same network as SCL:
   "rdeca_levo_zgoraj" := ("stevec_trenutno_s" = 0) AND "kljuc";
END_REGION

REGION Network 15: prizig lucke roka
   RUNG wire#powerrail
      { S7_Templates := "SrcType := Int" } EQ_Contact(in1 := "stevec_trenutno_s", in2 := 1)
      Contact( "kljuc" )
      Coil( "rdeca_desno_zgoraj" )
   END_RUNG
   // the same network as SCL:
   "rdeca_desno_zgoraj" := ("stevec_trenutno_s" = 1) AND "kljuc";
END_REGION

REGION Network 16: prizig lucke dvig
   RUNG wire#powerrail
      { S7_Templates := "SrcType := Int" } EQ_Contact(in1 := "stevec_trenutno_s", in2 := 2)
      Contact( "kljuc" )
      Coil( "rumena_levo_spodaj" )
   END_RUNG
   // the same network as SCL:
   "rumena_levo_spodaj" := ("stevec_trenutno_s" = 2) AND "kljuc";
END_REGION

REGION Network 17: prizig lucke prijemalo
   RUNG wire#powerrail
      { S7_Templates := "SrcType := Int" } EQ_Contact(in1 := "stevec_trenutno_s", in2 := 3)
      Contact( "kljuc" )
      Coil( "rumena_desno_spodaj" )
   END_RUNG
   // the same network as SCL:
   "rumena_desno_spodaj" := ("stevec_trenutno_s" = 3) AND "kljuc";
END_REGION
END_ORGANIZATION_BLOCK

(* ===== HMI "HMI_RT_1" =====
connection "HMI_Connection_1": ETHERNET, SIMATIC S7 300/400 MPI

HMI tags "Default tag table"
   "impulz_miza" : Bool = PLC "impulz_miza", 1 s
   "stevec_impulza_miza" : Int = PLC "stevec_impulza_miza", 100 ms
   "stevec_impulza_roka" : Int = PLC "stevec_impulza_roka", 100 ms
   "stevec_impulza_dvig" : Int = PLC "stevec_impulza_dvig", 100 ms
   "stevec_impulza_prijemalo" : Int = PLC "stevec_impulza_prijemalo", 100 ms
   "miza_smer" : Bool = PLC "miza_smer", 1 s
   "dvig_smer" : Bool = PLC "dvig_smer", 1 s
   "roka_smer" : Bool = PLC "roka_smer", 1 s
   "kljuc" : Bool = PLC "kljuc", 500 ms
   "Scada_Alarm_aktiven" : Bool, 1 s
   "Scada_Alarmi" : Word, 1 s
   "Scada_Potrjevanje_alarmov" : Bool, 1 s
   "Scada_miza_warning" : Bool, 1 s
   "Scada_roka_warning" : Bool, 1 s
   "Scada_dvig_warning" : Bool, 1 s
   "Scada_prijemalo_warning" : Bool, 1 s
   "recept" : Bool = PLC "recept", 1 s
   "Lokacije_Lokacija{0}_ID_lokacije" : Int, 1 s
   "Lokacije_Lokacija{1}_ID_lokacije" : Int, 1 s
   "Lokacije_Lokacija{2}_ID_lokacije" : Int, 1 s
   "Lokacije_Lokacija{3}_ID_lokacije" : Int, 1 s
   "Lokacije_Lokacija{4}_ID_lokacije" : Int, 1 s
   "Lokacije_Lokacija{5}_ID_lokacije" : Int, 1 s
   "Lokacije_Lokacija{6}_ID_lokacije" : Int, 1 s
   "Lokacije_Lokacija{7}_ID_lokacije" : Int, 1 s
   "Lokacije2_Lokacija2{0}_ID_lokacije" : Int, 1 s
   "Lokacije_Lokacija{0}_miza_lokacija" : Int, 1 s
   "Lokacije_Lokacija{0}_izteg_lokacija" : Int, 1 s
   "Lokacije_Lokacija{0}_stisk_lokacija" : Int, 1 s
   "Lokacije_Lokacija{0}_dvig_lokacija" : Int, 1 s
   "Lokacije_Lokacija{1}_miza_lokacija" : Int, 1 s
   "Lokacije_Lokacija{1}_izteg_lokacija" : Int, 1 s
   "Lokacije_Lokacija{1}_stisk_lokacija" : Int, 1 s
   "Lokacije_Lokacija{1}_dvig_lokacija" : Int, 1 s
   "Lokacije_Lokacija{2}_miza_lokacija" : Int, 1 s
   "Lokacije_Lokacija{2}_izteg_lokacija" : Int, 1 s
   "Lokacije_Lokacija{2}_stisk_lokacija" : Int, 1 s
   "Lokacije_Lokacija{2}_dvig_lokacija" : Int, 1 s
   "Lokacije_Lokacija{3}_miza_lokacija" : Int, 1 s
   "Lokacije_Lokacija{3}_izteg_lokacija" : Int, 1 s
   "Lokacije_Lokacija{3}_stisk_lokacija" : Int, 1 s
   "Lokacije_Lokacija{3}_dvig_lokacija" : Int, 1 s
   "Lokacije_Lokacija{4}_miza_lokacija" : Int, 1 s
   "Lokacije_Lokacija{4}_izteg_lokacija" : Int, 1 s
   "Lokacije_Lokacija{4}_stisk_lokacija" : Int, 1 s
   "Lokacije_Lokacija{4}_dvig_lokacija" : Int, 1 s
   "Lokacije_Lokacija{5}_miza_lokacija" : Int, 1 s
   "Lokacije_Lokacija{5}_izteg_lokacija" : Int, 1 s
   "Lokacije_Lokacija{5}_stisk_lokacija" : Int, 1 s
   "Lokacije_Lokacija{5}_dvig_lokacija" : Int, 1 s
   "Lokacije_Lokacija{6}_miza_lokacija" : Int, 1 s
   "Lokacije_Lokacija{6}_izteg_lokacija" : Int, 1 s
   "Lokacije_Lokacija{6}_stisk_lokacija" : Int, 1 s
   "Lokacije_Lokacija{6}_dvig_lokacija" : Int, 1 s
   "Lokacije_Lokacija{7}_miza_lokacija" : Int, 1 s
   "Lokacije_Lokacija{7}_izteg_lokacija" : Int, 1 s
   "Lokacije_Lokacija{7}_stisk_lokacija" : Int, 1 s
   "Lokacije_Lokacija{7}_dvig_lokacija" : Int, 1 s
   "Lokacije2_Lokacija2{0}_miza_lokacija" : Int, 1 s
   "Lokacije2_Lokacija2{0}_izteg_lokacija" : Int, 1 s
   "Lokacije2_Lokacija2{0}_stisk_lokacija" : Int, 1 s
   "Lokacije2_Lokacija2{0}_dvig_lokacija" : Int, 1 s
   "Lokacije2_Lokacija2{1}_miza_lokacija" : Int, 1 s
   "Lokacije2_Lokacija2{1}_izteg_lokacija" : Int, 1 s
   "Lokacije2_Lokacija2{1}_stisk_lokacija" : Int, 1 s
   "Lokacije2_Lokacija2{1}_dvig_lokacija" : Int, 1 s
   "Lokacije2_Lokacija2{2}_miza_lokacija" : Int, 1 s
   "Lokacije2_Lokacija2{2}_izteg_lokacija" : Int, 1 s
   "Lokacije2_Lokacija2{2}_stisk_lokacija" : Int, 1 s
   "Lokacije2_Lokacija2{2}_dvig_lokacija" : Int, 1 s
   "Lokacije2_Lokacija2{3}_miza_lokacija" : Int, 1 s
   "Lokacije2_Lokacija2{3}_izteg_lokacija" : Int, 1 s
   "Lokacije2_Lokacija2{3}_stisk_lokacija" : Int, 1 s
   "Lokacije2_Lokacija2{3}_dvig_lokacija" : Int, 1 s
   "Lokacije2_Lokacija2{4}_miza_lokacija" : Int, 1 s
   "Lokacije2_Lokacija2{4}_izteg_lokacija" : Int, 1 s
   "Lokacije2_Lokacija2{4}_stisk_lokacija" : Int, 1 s
   "Lokacije2_Lokacija2{4}_dvig_lokacija" : Int, 1 s
   "Lokacije2_Lokacija2{5}_miza_lokacija" : Int, 1 s
   "Lokacije2_Lokacija2{5}_izteg_lokacija" : Int, 1 s
   "Lokacije2_Lokacija2{5}_stisk_lokacija" : Int, 1 s
   "Lokacije2_Lokacija2{5}_dvig_lokacija" : Int, 1 s
   "Lokacije2_Lokacija2{6}_miza_lokacija" : Int, 1 s
   "Lokacije2_Lokacija2{6}_izteg_lokacija" : Int, 1 s
   "Lokacije2_Lokacija2{6}_stisk_lokacija" : Int, 1 s
   "Lokacije2_Lokacija2{6}_dvig_lokacija" : Int, 1 s
   "Lokacije2_Lokacija2{7}_miza_lokacija" : Int, 1 s
   "Lokacije2_Lokacija2{7}_izteg_lokacija" : Int, 1 s
   "Lokacije2_Lokacija2{7}_stisk_lokacija" : Int, 1 s
   "Lokacije2_Lokacija2{7}_dvig_lokacija" : Int, 1 s
   "miza_premik" : Bool = PLC "miza_premik", 1 s
   "dvig_premik" : Bool = PLC "dvig_premik", 1 s
   "roka_premik" : Bool = PLC "roka_premik", 1 s
   "prijemalo_premik" : Bool = PLC "prijemalo_premik", 1 s

discrete alarms
   1: '', class Warnings, trigger "Scada_Alarmi" bit 8
   2: '', class Warnings, trigger "Scada_Alarmi" bit 9
   3: '', class Warnings, trigger "Scada_Alarmi" bit 10
   4: '', class Warnings, trigger "Scada_Alarmi" bit 11
   5: '', class Errors, trigger "Scada_Alarmi" bit 12
   6: '', class Errors, trigger "Scada_Alarmi" bit 13
   7: '', class Errors, trigger "Scada_Alarmi" bit 14
   8: '', class Errors, trigger "Scada_Alarmi" bit 15
   9: '', class Info, trigger "Scada_Alarmi" bit 0
   10: '', class Info, trigger "Scada_Alarmi" bit 1

recipe "Recept": miza0 <- "Lokacije_Lokacija{0}_miza_lokacija", izteg0 <- "Lokacije_Lokacija{0}_izteg_lokacija", stisk0 <- "Lokacije_Lokacija{0}_stisk_lokacija", dvig0 <- "Lokacije_Lokacija{0}_dvig_lokacija", miza1 <- "Lokacije_Lokacija{1}_miza_lokacija", izteg1 <- "Lokacije_Lokacija{1}_izteg_lokacija", stisk1 <- "Lokacije_Lokacija{1}_stisk_lokacija", dvig1 <- "Lokacije_Lokacija{1}_dvig_lokacija", miza2 <- "Lokacije_Lokacija{2}_miza_lokacija", izteg2 <- "Lokacije_Lokacija{2}_izteg_lokacija", stisk2 <- "Lokacije_Lokacija{2}_stisk_lokacija", dvig2 <- "Lokacije_Lokacija{2}_dvig_lokacija", miza3 <- "Lokacije_Lokacija{3}_miza_lokacija", izteg3 <- "Lokacije_Lokacija{3}_izteg_lokacija", stisk3 <- "Lokacije_Lokacija{3}_stisk_lokacija", dvig3 <- "Lokacije_Lokacija{3}_dvig_lokacija", miza4 <- "Lokacije_Lokacija{4}_miza_lokacija", izteg4 <- "Lokacije_Lokacija{4}_izteg_lokacija", stisk4 <- "Lokacije_Lokacija{4}_stisk_lokacija", dvig4 <- "Lokacije_Lokacija{4}_dvig_lokacija", miza5 <- "Lokacije_Lokacija{5}_miza_lokacija", izteg5 <- "Lokacije_Lokacija{5}_izteg_lokacija", stisk5 <- "Lokacije_Lokacija{5}_stisk_lokacija", dvig5 <- "Lokacije_Lokacija{5}_dvig_lokacija", miza6 <- "Lokacije_Lokacija{6}_miza_lokacija", izteg6 <- "Lokacije_Lokacija{6}_izteg_lokacija", stisk6 <- "Lokacije_Lokacija{6}_stisk_lokacija", dvig6 <- "Lokacije_Lokacija{6}_dvig_lokacija", miza7 <- "Lokacije_Lokacija{7}_miza_lokacija", izteg7 <- "Lokacije_Lokacija{7}_izteg_lokacija", stisk7 <- "Lokacije_Lokacija{7}_stisk_lokacija", dvig7 <- "Lokacije_Lokacija{7}_dvig_lokacija"

recipe "Recept2": miza0 <- "Lokacije2_Lokacija2{0}_miza_lokacija", izteg0 <- "Lokacije2_Lokacija2{0}_izteg_lokacija", stisk0 <- "Lokacije2_Lokacija2{0}_stisk_lokacija", dvig0 <- "Lokacije2_Lokacija2{0}_dvig_lokacija", miza1 <- "Lokacije2_Lokacija2{1}_miza_lokacija", izteg1 <- "Lokacije2_Lokacija2{1}_izteg_lokacija", stisk1 <- "Lokacije2_Lokacija2{1}_stisk_lokacija", dvig1 <- "Lokacije2_Lokacija2{1}_dvig_lokacija", miza2 <- "Lokacije2_Lokacija2{2}_miza_lokacija", izteg2 <- "Lokacije2_Lokacija2{2}_izteg_lokacija", stisk2 <- "Lokacije2_Lokacija2{2}_stisk_lokacija", dvig2 <- "Lokacije2_Lokacija2{2}_dvig_lokacija", miza3 <- "Lokacije2_Lokacija2{3}_miza_lokacija", izteg3 <- "Lokacije2_Lokacija2{3}_izteg_lokacija", stisk3 <- "Lokacije2_Lokacija2{3}_stisk_lokacija", dvig3 <- "Lokacije2_Lokacija2{3}_dvig_lokacija", miza4 <- "Lokacije2_Lokacija2{4}_miza_lokacija", izteg4 <- "Lokacije2_Lokacija2{4}_izteg_lokacija", stisk4 <- "Lokacije2_Lokacija2{4}_stisk_lokacija", dvig4 <- "Lokacije2_Lokacija2{4}_dvig_lokacija", miza5 <- "Lokacije2_Lokacija2{5}_miza_lokacija", izteg5 <- "Lokacije2_Lokacija2{5}_izteg_lokacija", stisk5 <- "Lokacije2_Lokacija2{5}_stisk_lokacija", dvig5 <- "Lokacije2_Lokacija2{5}_dvig_lokacija", miza6 <- "Lokacije2_Lokacija2{6}_miza_lokacija", izteg6 <- "Lokacije2_Lokacija2{6}_izteg_lokacija", stisk6 <- "Lokacije2_Lokacija2{6}_stisk_lokacija", dvig6 <- "Lokacije2_Lokacija2{6}_dvig_lokacija", miza7 <- "Lokacije2_Lokacija2{7}_miza_lokacija", izteg7 <- "Lokacije2_Lokacija2{7}_izteg_lokacija", stisk7 <- "Lokacije2_Lokacija2{7}_stisk_lokacija", dvig7 <- "Lokacije2_Lokacija2{7}_dvig_lokacija"

Template "Template_1" 640x480
   Button "Template_Button_Glavni_zaslon" at 117,402 size 127x51
   Button "Template_Button_1" at 267,402 size 127x51
   Button "Template_Button_2" at 413,402 size 127x51
   DateTimeField "Template_Date/time field_1" at 133,5 size 359x27

screen "OsnovniZaslon" 640x480, template "Template_1"
   IOField "I/O field_1" at 93,81 size 67x32
   TextField "Text field_1" at 82,52 size 98x22
   IOField "I/O field_2" at 214,81 size 67x32
   TextField "Text field_2" at 200,52 size 101x22
   TextField "Text field_3" at 324,52 size 97x22
   TextField "Text field_4" at 445,52 size 135x22
   IOField "I/O field_3" at 339,81 size 67x32
   IOField "I/O field_4" at 465,81 size 67x32
   TextField "Text field_5" at 445,122 size 115x22
   SymbolLibrary "Symbol library_1" at 82,122 size 37x26
   SymbolLibrary "Symbol library_2" at 133,122 size 37x26
   SymbolLibrary "Symbol library_3" at 347,122 size 26x37
   SymbolLibrary "Symbol library_4" at 373,122 size 26x37
   SymbolLibrary "Symbol library_5" at 200,122 size 37x26
   SymbolLibrary "Symbol library_6" at 255,122 size 37x26
   TextField "Text field_6" at 51,183 size 97x28
   TextField "Text field_7" at 51,278 size 139x28
   TextField "Text field_8" at 458,183 size 84x28
   TextField "Text field_9" at 446,220 size 40x22
   TextField "Text field_10" at 513,219 size 43x22
   TextField "Text field_11" at 447,284 size 39x22
   TextField "Text field_12" at 513,284 size 43x22

screen "Alarmi" 640x480, template "Template_1"
   AlarmView "Alarm view_1" at 81,109 size 462x259
   Button "Button_1" at 351,57 size 180x32

screen "Recepti" 640x480, template "Template_1"
   RecipeView "Recipe view_1" at 109,78 size 404x310
   Switch "Switch_1" at 369,45 size 99x27
   TextField "Text field_1" at 180,45 size 180x22
*)